// ---- DUTs/Controllers/Band.TcPOU
FUNCTION Band : LREAL
VAR_INPUT
	Value: lreal;
	Target: LREAL;
	Width: LREAL;
END_VAR
VAR
END_VAR

  Band := LimitValue(Value - Target, -Width, Width) / Width;

END_FUNCTION

// ---- DUTs/Controllers/BandLimit.TcPOU
FUNCTION BandLimit : LREAL
VAR_INPUT
	Value: LREAL;
	Target: LREAL;
	Width: LREAL;
	MinValue: LREAL;
	MaxValue: LREAL;
END_VAR
VAR
END_VAR

BandLimit := LimitValue(Band(Value, Target, Width), MinValue, MaxValue);

END_FUNCTION

// ---- DUTs/Controllers/Controller.TcPOU
FUNCTION_BLOCK Controller
VAR_INPUT
	EN: BOOL;
    SP: LREAL;          (* Set point                           *)
    PV: LREAL;          (* Process value                       *)
    p_gain: LREAL;      (* Proportional gain (stiffness)       *)
    i_gain: LREAL;      (* integral gain (windup)              *)
END_VAR
VAR_OUTPUT
	ENO: BOOL;
    CV: LREAL;          (* Control value              *)
END_VAR
VAR
    { Parameters }

    { Calculated values }

    { Local variables}
    integral: LREAL;
    last_error: LREAL;
    last_output: LREAL;
    this_target: LREAL;
    next_target: LREAL;
    ITimer: Timer;    (* Integration timer *)
    LastITime: LINT;
    Timer: Timer;    (* Update timer *)
    MinControl: Timer;
    MaxControl: Timer;
END_VAR

ENO := EN;
IF EN THEN
	Compute();
ELSE
	Reset();	
END_IF

METHOD Compute : BOOL
VAR_INPUT
END_VAR
VAR
  this_error: LREAL;
  this_output: LREAL;
  new_integral: LREAL;
  TimeValue: LINT;

END_VAR
(* the desired PV for this iteration is the value     *)
(* calculated as next_target during the last loop     *)
this_target := next_target;

next_target := SP;

(* the error for the current pass is the difference   *)
(* between the current target and the current PV      *)
this_error := this_target - PV;

{ the new error is added to the integral             }
TimeValue := ITimer.ElapsedTime();
new_integral := integral + i_gain * (this_target - PV) * ((1.0 * LINT_TO_LREAL(TimeValue - LastITime)) / LINT_TO_LREAL(ITimer.TimeoutTime));
LastITime := TimeValue;
IF (new_integral + p_gain * this_error) > 1 THEN
	integral := 1 - p_gain * this_error;
ELSIF (new_integral + p_gain * this_error) < 0 THEN
	integral := -p_gain * this_error;
ELSE
	integral := new_integral;
END_IF;
IF ITimer.Timeout() THEN
	ITimer.Restart();
	LastITime := 0;
END_IF;

(* now that all of the variable terms have been       *)
(* computed they can be multiplied by the appropriate *)
(* coefficients and the resulting products summed     *)
this_output := p_gain * this_error + integral;

last_error := this_error;

(* now check the output value for absolute limits     *)
IF (this_output < 0) THEN
	(* Limit I *)
	if integral < 0 then
		integral := LimitValue(integral, integral - this_output, 0);
	END_IF;
	this_output := 0;
ELSIF (this_output > 1) THEN
	(* Limit I *)
	if integral > 0 then
		integral := LimitValue(integral, 0, integral - (this_output - 1));
	END_IF;
	(* Limit output *)
	this_output := 1;
END_IF;

(* store the new output value to be used as the old   *)
(* output value on the next loop pass                 *)
last_output := this_output;

CV := this_output;
IF Timer.Timeout() THEN
	Timer.Restart();
END_IF;
IF CV > 0.01 THEN
	MinControl.Restart();
END_IF;
IF CV < (1 - 0.01) THEN
	MaxControl.Restart();
END_IF;
END_METHOD

METHOD FB_init : BOOL
VAR_INPUT
	bInitRetains : BOOL; // if TRUE, the retain variables are initialized (warm start / cold start)
	bInCopyCode : BOOL;  // if TRUE, the instance afterwards gets moved into the copy code (online change)
END_VAR
p_gain := 0.5;
i_gain := 0.5;
ITimer.TimeoutTime := 30000;
Timer.TimeoutTime := 1000;
END_METHOD

METHOD Preset : BOOL
VAR_INPUT
	Target: LREAL;
	Control: LREAL;
END_VAR
  last_error := 0;
  last_output := Control;
  next_target := Target;
  this_target := Target;
  ResetIntegral();
  integral := Control;
  CV := Control;
  SP := Target;
END_METHOD

METHOD Reset : BOOL
VAR_INPUT
END_VAR
  ResetIntegral();
  last_error := 0;
  last_output := 0;
  next_target := 0;
  this_target := 0;
  CV := 0;
  SP := 0;
  MinControl.Restart();
  MaxControl.Restart();
END_METHOD

METHOD ResetIntegral : BOOL
VAR_INPUT
END_VAR
  integral := 0;
  ITimer.Restart();
  LastITime := ITimer.ElapsedTime();
END_METHOD

END_FUNCTION_BLOCK

// ---- DUTs/Controllers/InterpolateNewton.TcPOU
FUNCTION_BLOCK InterpolateNewton
VAR_INPUT
	EN: BOOL;
	x: LREAL;
END_VAR
VAR_OUTPUT
	ENO: BOOL;
	y: LREAL;
END_VAR
VAR CONSTANT
	NUM_POINTS: INT := 9;
END_VAR
VAR
	InitDone: BOOL;
	yd: ARRAY [0..NUM_POINTS - 1, 0..NUM_POINTS - 1] OF LREAL;
	i: INT;
END_VAR
VAR PERSISTENT
	xd: ARRAY [0..NUM_POINTS - 1] OF LREAL;
	yv: ARRAY [0..NUM_POINTS - 1] OF LREAL;
END_VAR

IF NOT InitDone THEN
	FOR i := 0 TO NUM_POINTS - 1 DO
		yd[i, 0] := yv[i];
	END_FOR
	DividedDiffTable();
	InitDone := TRUE;
END_IF
y := ApplyFormula(x);
ENO := EN;

METHOD ApplyFormula : LREAL
VAR_INPUT
	Value: LREAL;
END_VAR
VAR
	Sum: LREAL;
	i: INT;
END_VAR
Sum := yd[0, 0];
FOR i := 1 TO NUM_POINTS - 1 DO
	Sum := Sum + ProTerm(i, Value) * yd[0, i];
END_FOR
ApplyFormula := Sum;
END_METHOD

METHOD DividedDiffTable : BOOL
VAR_INPUT
END_VAR
VAR
	i: INT;
	j: int;
END_VAR
FOR i := 1 TO NUM_POINTS - 1 DO
	FOR j := 0 TO NUM_POINTS - i - 1 DO
		IF ABS(xd[j] - xd[i + j]) > 0.00000001 THEN
			yd[j,i] := (yd[j,i - 1] - yd[j + 1,i - 1]) / (xd[j] - xd[i + j]);			
		END_IF
	END_FOR
END_FOR
DividedDiffTable := TRUE;
END_METHOD

METHOD ProTerm : LREAL
VAR_INPUT
	i: INT;
	Value: LREAL;
END_VAR
VAR
	Pro: LREAL;
	j: int;
END_VAR
Pro := 1;
FOR j := 0 TO i - 1 DO
	Pro := Pro * (Value - xd[j]);
END_FOR
ProTerm := Pro;
END_METHOD

END_FUNCTION_BLOCK

// ---- DUTs/Controls/ExtractAirControl.TcPOU
FUNCTION_BLOCK ExtractAirControl
VAR_INPUT
	EN: BOOL;
END_VAR
VAR_OUTPUT
	ENO: BOOL;
END_VAR
VAR
END_VAR

ENO := EN;

END_FUNCTION_BLOCK

// ---- DUTs/Fire/FireDamper.TcPOU
FUNCTION_BLOCK FireDamper EXTENDS Damper
VAR_INPUT
END_VAR
VAR_OUTPUT
END_VAR
VAR
END_VAR

END_FUNCTION_BLOCK

// ---- DUTs/Fire/SmokeDetector.TcPOU
FUNCTION_BLOCK SmokeDetector
VAR_INPUT
	EN: BOOL;
	Input: REFERENCE TO AnalogInput;
	FireAlarm: REFERENCE TO AnalogAlarm;
	ServiceAlarm: REFERENCE TO AnalogAlarm;
END_VAR
VAR_OUTPUT
	ENO: BOOL;
END_VAR
VAR
END_VAR

END_FUNCTION_BLOCK

// ---- DUTs/GreenMaster/IO/GreenMasterAIU.TcPOU
FUNCTION_BLOCK GreenMasterAIU EXTENDS GreenMasterAIU_Base
VAR_INPUT
END_VAR
VAR_OUTPUT
END_VAR
VAR
	IO_AI_09: PressureInput;
	IO_AI_10: PressureInput;
	IO_AI_11: PressureInput;
	IO_AI_12: PressureInput;
	IO_AI_13: PressureInput;
	IO_AI_14: PressureInput;
	IO_AI_15: PressureInput;
	IO_AI_16: PressureInput;
END_VAR


// PAGE AI
IO_AI_09(ProcessError := Globals.IO.AIn.AI17_Error, ProcessValue := Globals.IO.AIn.AI17, Range := 3500); // PressureInput
T_BF1_Error := IO_AI_09.Error;
IO_AI_10(ProcessError := Globals.IO.AIn.AI18_Error, ProcessValue := Globals.IO.AIn.AI18, Range := 3500); // PressureInput
T_BF1 := IO_AI_09.Value;
F_BF1_Error := IO_AI_10.Error;
F_BF1 := IO_AI_10.Value;
IO_AI_11(ProcessError := Globals.IO.AIn.AI19_Error, ProcessValue := Globals.IO.AIn.AI19, Range := 500); // PressureInput
T_BP2_Error := IO_AI_11.Error;
IO_AI_12(ProcessError := Globals.IO.AIn.AI20_Error, ProcessValue := Globals.IO.AIn.AI20, Range := 500); // PressureInput
T_BP2 := IO_AI_11.Value;
F_BP2_Error := IO_AI_12.Error;
F_BP2 := IO_AI_12.Value;
IO_AI_13(ProcessError := Globals.IO.AIn.AI21_Error, ProcessValue := Globals.IO.AIn.AI21, Range := 500); // PressureInput
F_BP3_Error := IO_AI_13.Error;
IO_AI_14(ProcessError := Globals.IO.AIn.AI22_Error, ProcessValue := Globals.IO.AIn.AI22, Range := 500); // PressureInput
F_BP3 := IO_AI_13.Value;
T_BP1_Error := IO_AI_14.Error;
T_BP1 := IO_AI_14.Value;
IO_AI_15(ProcessError := Globals.IO.AIn.AI23_Error, ProcessValue := Globals.IO.AIn.AI23, Range := 500); // PressureInput
F_BP1_Error := IO_AI_15.Error;
IO_AI_16(ProcessError := Globals.IO.AIn.AI24_Error, ProcessValue := Globals.IO.AIn.AI24); // PressureInput
F_BP1 := IO_AI_15.Value;

END_FUNCTION_BLOCK

// ---- DUTs/IO/AnalogSwitch.TcPOU
FUNCTION_BLOCK AnalogSwitch
VAR_INPUT
	EN: BOOL;
	Index: INT;
	Input01: LREAL;
	Input02: LREAL;
	Input03: LREAL;
	Input04: LREAL;
	Input05: LREAL;
	Input06: LREAL;
	Input07: LREAL;
	Input08: LREAL;
END_VAR
VAR_OUTPUT
	ENO: BOOL;
	Output: LREAL;
END_VAR
VAR
END_VAR

END_FUNCTION_BLOCK

// ---- DUTs/ModbusRTU/ModbusWriteWord.TcPOU
FUNCTION_BLOCK ModbusWriteWord EXTENDS ModbusIo
VAR_INPUT
	Value: WORD;
END_VAR
VAR_OUTPUT
END_VAR
VAR
END_VAR

SUPER^();

END_FUNCTION_BLOCK

// ---- DUTs/Parameters/Regulation/DefaultParametersFB.TcPOU
FUNCTION_BLOCK DefaultParametersFB
VAR_INPUT
END_VAR
VAR_OUTPUT
END_VAR
VAR
END_VAR

END_FUNCTION_BLOCK

// ---- DUTs/Parameters/Simulation/SimulateFlow.TcPOU
FUNCTION_BLOCK SimulateFlow
VAR_INPUT
	EN: BOOL;
	SP: LREAL;
	CV: LREAL;
END_VAR
VAR_OUTPUT
	ENO: BOOL;
	Flow: LREAL;
END_VAR
VAR
	Ramp: Ramp;
	FlowFactor: LREAL;
END_VAR

IF EN THEN
	FlowFactor := 1;
	FlowFactor := FlowFactor * MAX(1, CV / 500);
	Ramp(Target := SP * 30000, SpeedUp := 50, SpeedDown := 100, Value => Flow);
END_IF

END_FUNCTION_BLOCK

// ---- DUTs/Parameters/Simulation/SimulationParametersFB.TcPOU
FUNCTION_BLOCK SimulationParametersFB
VAR_INPUT
END_VAR
VAR_OUTPUT
END_VAR
VAR
END_VAR

SimCounter := SimCounter + 1;

END_FUNCTION_BLOCK

// ---- DUTs/Parameters/System/Exercise/ExerciseExternalFireControlParametersFB.TcPOU
FUNCTION_BLOCK ExerciseExternalFireControlParametersFB
VAR_INPUT
END_VAR
VAR_OUTPUT
END_VAR
VAR
END_VAR

END_FUNCTION_BLOCK

// ---- DUTs/Parameters/System/Operation/TimeChannelDayParametersFB.TcPOU
FUNCTION_BLOCK TimeChannelDayParametersFB
VAR_INPUT
END_VAR
VAR_OUTPUT
END_VAR
VAR
END_VAR

END_FUNCTION_BLOCK

// ---- DUTs/System/Supervisor.TcPOU
FUNCTION_BLOCK Supervisor
VAR_INPUT
	EN: BOOL;
	Stop: BOOL;
END_VAR
VAR_OUTPUT
	ENO: BOOL;
END_VAR
VAR
END_VAR
VAR PERSISTENT
END_VAR

ENO := EN AND NOT Stop;

METHOD FB_init : BOOL
VAR_INPUT
	bInitRetains : BOOL; // if TRUE, the retain variables are initialized (warm start / cold start)
	bInCopyCode : BOOL;  // if TRUE, the instance afterwards gets moved into the copy code (online change)
END_VAR
END_METHOD

END_FUNCTION_BLOCK

// ---- DUTs/Utilities/ActuatorMonitor.TcPOU
FUNCTION_BLOCK ActuatorMonitor
VAR_INPUT
	Output: LREAL;
	Input: LREAL;
	Activated: BOOL := TRUE;
	ActivatedError: BOOL := FALSE;
	TimeoutMs: DINT := 30000;
	Treshold: LREAL := 0.1;
END_VAR
VAR_OUTPUT
	Error: BOOL := FALSE;
END_VAR
VAR
	ActivatedSignal: DigitalSignal;
	OutputOnTimer: Timer;
	InputOffTimer: Timer;
END_VAR

// Measure ON time for activation signal
ActivatedSignal(Signal := Activated);

// Measure ON time for output signal
IF Output < Treshold THEN
	OutputOnTimer.Restart();
END_IF

// Measure OFF time for 50% input signal
IF Input >= (Treshold / 2) THEN
	InputOffTimer.Restart();
END_IF

Error := 	(
				(ActivatedSignal.OnTime() > TimeoutMs) AND 
				(OutputOnTimer.ElapsedTime() > TimeoutMs) AND 
				(
					(InputOffTimer.ElapsedTime() > TimeoutMs) OR
					ActivatedError
				)
			);

END_FUNCTION_BLOCK

// ---- DUTs/Utilities/AnalogMultiplexer.TcPOU
FUNCTION_BLOCK AnalogMultiplexer
VAR_INPUT
	bSelect: BOOL;
	iSelect: INT := -1;
	In0: LREAL := 0;
	In1: LREAL := 0;
	In2: LREAL := 0;
	In3: LREAL := 0;
END_VAR
VAR_OUTPUT
	Out: LREAL;
END_VAR
VAR
END_VAR

IF iSelect = -1 THEN
	IF bSelect THEN
		Out := In1;
	ELSE
		Out := In0;
	END_IF
ELSE
	CASE iSelect OF
		0: 	Out := In0;
		1: 	Out := In1;
		2: 	Out := In2;
		3: 	Out := In3;
	END_CASE
END_IF

END_FUNCTION_BLOCK

// ---- DUTs/Utilities/ifc_int.TcPOU
FUNCTION ifc_int : INT
VAR_INPUT
	Condition: BOOL;
	ValueTrue: INT;
	ValueFalse: INT;
END_VAR
VAR
END_VAR

IF Condition THEN
	ifc_int := ValueTrue;
ELSE
	ifc_int := ValueFalse;
END_IF

END_FUNCTION

// ---- DUTs/Utilities/BOOL_BMUX.TcPOU
FUNCTION BOOL_BMUX : BOOL
VAR_INPUT
	B: BOOL;
	X: BOOL;
	Y: BOOL
;
END_VAR
VAR
END_VAR

IF NOT B THEN
	BOOL_BMUX := X;
ELSE
	BOOL_BMUX := Y;
END_IF

END_FUNCTION

// ---- DUTs/Utilities/EMA.TcPOU
FUNCTION_BLOCK EMA
VAR_INPUT
	NewValue: LREAL;
END_VAR
VAR_OUTPUT
	Value: LREAL;
END_VAR
VAR
	Weight: LREAL;
END_VAR

Value := Weight * NewValue + (1 - Weight) * Value;

METHOD FB_init : BOOL
VAR_INPUT
	bInitRetains : BOOL; // if TRUE, the retain variables are initialized (warm start / cold start)
	bInCopyCode : BOOL;  // if TRUE, the instance afterwards gets moved into the copy code (online change)
END_VAR
SetSampleCount(100);
END_METHOD

METHOD SetSampleCount : BOOL
VAR_INPUT
	n: int;
END_VAR
Weight := 2.0 / (1.0 + n);
END_METHOD

METHOD SetValue : BOOL
VAR_INPUT
	NewValue: LREAL;
END_VAR
Value := NewValue;
END_METHOD

END_FUNCTION_BLOCK

// ---- DUTs/Utilities/GetBit.TcPOU
FUNCTION GetBit : BOOL
VAR_INPUT
	Value: ULINT;
	BitNr: INT;
END_VAR
VAR
END_VAR

GetBit := (Value AND SHL(INT_TO_ULINT(1), BitNr)) <> 0;

END_FUNCTION

// ---- DUTs/Utilities/PulseCounter.TcPOU
FUNCTION_BLOCK PulseCounter
VAR_INPUT
	FM: BOOL;
END_VAR
VAR_OUTPUT
	Flow: LREAL;
	PulseCounter: LINT;
END_VAR
VAR
	Tmp: BOOL;
	Now: LINT;
	Last_FM: BOOL;
	LastTime: LINT;
	FilteredFlow: EMA;
	Pulse: BOOL;
	LastPulseLength: LINT;
END_VAR

Tmp := FM;
Now := GetTickCount();
Pulse := (Tmp AND (Tmp <> Last_FM)); 
IF Pulse THEN
	PulseCounter := PulseCounter + 1;
	LastPulseLength := Now - LastTime;
	IF (Now - LastTime) > 0 THEN
		FilteredFlow(NewValue := 3.6 / (LINT_TO_LREAL(Now - LastTime) / 1000.0));
	END_IF
	LastTime := Now;
END_IF
Last_FM := Tmp;
IF (Now - LastTime) > (2 * LastPulseLength) THEN
	IF (Now - LastTime) > 0 THEN
		FilteredFlow(NewValue := 3.6 / (LINT_TO_LREAL(Now - LastTime) / 1000.0));
	END_IF
END_IF
IF (Now - LastTime) > 30000 THEN
	FilteredFlow.SetValue(0);
END_IF
Flow := FilteredFlow.Value;

METHOD FB_init : BOOL
VAR_INPUT
	bInitRetains : BOOL; // if TRUE, the retain variables are initialized (warm start / cold start)
	bInCopyCode : BOOL;  // if TRUE, the instance afterwards gets moved into the copy code (online change)
END_VAR
FilteredFlow.SetSampleCount(5);
END_METHOD

END_FUNCTION_BLOCK

// ---- DUTs/Utilities/PWM.TcPOU
FUNCTION_BLOCK PWM
VAR_INPUT
END_VAR
VAR_OUTPUT
END_VAR
VAR
	Timer: Timer;
	CurrentDutyCycle: LREAL;
	FPeriod: LREAL;
	FDutyCycle: LREAL;
	FMinValue: LREAL := 0.05; // 5% / 95% min/max value	
END_VAR

PROPERTY DutyCycle : LREAL
GET
DutyCycle := CurrentDutyCycle;
END_GET
SET
VAR
	TimeValue: lreal;	
END_VAR
TimeValue := DutyCycle * Period;
IF (TimeValue < MinValue) THEN
	FDutyCycle := 0;
ELSIF (TimeValue > (Period - MinValue)) THEN
	FDutyCycle := 1;
else
	FDutyCycle := DutyCycle;
END_IF
END_SET
END_PROPERTY

PROPERTY MinValue : LREAL
GET
MinValue := FMinValue;
END_GET
SET
FMinValue := MinValue;
END_SET
END_PROPERTY

PROPERTY Period : LREAL
GET
Period := FPeriod;
END_GET
SET
IF FPeriod <> Period THEN
	FPeriod := Period;
	CurrentDutyCycle := DutyCycle;
	Timer.Restart();
END_IF;
END_SET
END_PROPERTY

METHOD State : BOOL
VAR_INPUT
END_VAR
VAR
	ElapsedTime: LINT;
	Res: BOOL;
END_VAR
ElapsedTime := Timer.ElapsedTime();
IF (ElapsedTime > LREAL_TO_LINT(Period * 1000)) THEN
	ElapsedTime := TRUNC(Period * 1000);
END_IF
Res := ElapsedTime <= LREAL_TO_LINT(CurrentDutyCycle * Period * 1000);
IF (ElapsedTime >= LREAL_TO_LINT(Period * 1000)) THEN
	Timer.Restart();
	CurrentDutyCycle := FDutyCycle;
END_IF;
State := Res;
END_METHOD

END_FUNCTION_BLOCK

// ---- DUTs/Utilities/LREAL_TO_WORD_SAFE.TcPOU
FUNCTION LREAL_TO_WORD_SAFE : WORD
VAR_INPUT
	Value: LREAL;
END_VAR
VAR
END_VAR

LREAL_TO_WORD_SAFE := TO_WORD(TO_LINT(Value));

END_FUNCTION

// ---- DUTs/Utilities/SetBit.TcPOU
FUNCTION SetBit : ULINT
VAR_INPUT
	Value: ULINT;
	BitNr: INT;
	State: BOOL;
END_VAR
VAR
END_VAR

IF State THEN
	SetBit := (Value AND (NOT SHL(INT_TO_ULINT(1), BitNr))) OR SHL(INT_TO_ULINT(1), BitNr);
ELSE
	SetBit := (Value AND (NOT SHL(INT_TO_ULINT(1), BitNr)));
END_IF

END_FUNCTION

// ---- DUTs/Valves/BaseValve.TcPOU
FUNCTION_BLOCK BaseValve
VAR_INPUT
	Open: REFERENCE TO BOOL;
	IsOpen: REFERENCE TO BOOL;
	IsClosed: REFERENCE TO BOOL;
END_VAR
VAR_OUTPUT
END_VAR
VAR
END_VAR

END_FUNCTION_BLOCK

// ---- DUTs/Valves/Valve.TcPOU
FUNCTION_BLOCK Valve EXTENDS BaseValve
VAR_INPUT
	IO_Open: REFERENCE TO DigitalOutput;
	IO_FB1, IO_FB2: REFERENCE TO DigitalInput;
END_VAR
VAR_OUTPUT
END_VAR
VAR
	ValveMonitor: ValveMonitor; 
	Error: BOOL;
END_VAR

ValveMonitor(Valve := Open, FB1 := IsOpen, FB2 := IsClosed);
Error := ValveMonitor.Error;

END_FUNCTION_BLOCK

// ---- DUTs/Valves/ValveMonitor.TcPOU
FUNCTION_BLOCK ValveMonitor
VAR_INPUT
	Valve: BOOL;	// Valve DO
	FB1: BOOL;		// Open DI
	FB2: BOOL;		// Closed DI
	Timeout: TIME;
END_VAR
VAR_OUTPUT
	Error: BOOL;
END_VAR
VAR
	ValveSignal: DigitalSignal;
	ValveOpenTimer: Timer;
	ValveClosedTimer: Timer;
END_VAR

ValveSignal(Signal := Valve);
IF Main.GreenMaster.GetParameters().System.Operation.State <> SystemStates.Run THEN
	Error := FALSE;
ELSE
	Error := ((ValveSignal.OnTime() > TO_LINT(T#30S)) AND (NOT FB1)) OR
		((ValveSignal.OffTime() > TO_LINT(T#30S)) AND (NOT FB2));	
END_IF

END_FUNCTION_BLOCK

// ---- DUTs/Ventilation/FB_GM_NIGHTCOOL.TcPOU
FUNCTION_BLOCK FB_GM_NIGHTCOOL
VAR_INPUT
	bDayOperation						: BOOL; // Normal daytime operation
	rNormalSAPressure					: REAL; // Normal daytime operation setpoint for supply air pressure
	rNormalEAPressure					: REAL; // Normal daytime operation setpoint for extract air pressure
	rNormalTemperature					: REAL; // Normal daytime operation setpoint for supply air temperature
END_VAR
VAR_OUTPUT
	bStartNightcool						: BOOL; // Starts GreenMaster in nightcool	
	rSAPressure							: REAL; // Supply air pressure when nightcooling is active
	rEAPressure							: REAL;	// Extract air pressure when nightcooling is active
	rSATemperature						: REAL; // Supply air temperature when nightcooling is active
	bNightCoolActive					: BOOL; // Nightcooling is active
	rExtractAirTemperature				: REAL;	// Saftey input
END_VAR
VAR PERSISTENT
	rSupplyPressure						: REAL; // Supply air pressure when nightcooling is active
	rExtractPressure					: REAL; // Extract air pressure when nightcooling is active
	rSupplyTemperature					: REAL; // Supply air temperature when nightcooling is active
	bCMD								: BOOL; // Start nightcooling from HMI
END_VAR

// Om vi kör nattkyla så har vi nya börvärden
IF bStartNightcool THEN
	rSAPressure := rSupplyPressure;   // New SA Pressure setpoint
	rEAPressure := rExtractPressure;  // New EA Pressire setpint
	rSATemperature :=  MAX (13,rSupplyTemperature); // New SA temperature setpoint with limit 
	bNightCoolActive :=TRUE;
ELSE
	rSAPressure := rNormalSAPressure;
    rEAPressure := rNormalEAPressure;
    rSATemperature := rNormalTemperature;
	bNightCoolActive :=FALSE;
END_IF

// Sätter utgång för att starta aggregat (med säkerhetsfunktion då frånluftstemperatur blir för låg)
IF NOT bDayOperation AND NOT(rExtractAirTemperature < 17) THEN
	IF bCMD THEN
		bStartNightcool := TRUE;
	ELSE
		bStartNightcool := FALSE;
	END_IF
ELSE 
	bStartNightcool := FALSE;
END_IF

END_FUNCTION_BLOCK

// ---- POUs/AdsWriteVariable.TcPOU
FUNCTION_BLOCK AdsWriteVariable
VAR_INPUT
	NetID: STRING := '';
	Name: STRING;
	EN: BOOL;
	Source: PVOID;
END_VAR
VAR_OUTPUT
	ENO: BOOL;
END_VAR
VAR
	PLC_ReadSymInfoByName: PLC_ReadSymInfoByName;
	ADSWRITE: ADSWRITE;
	State : INT := 0;
END_VAR

CASE State OF
0:
	IF EN THEN
		State := 1;
	END_IF
1:	
	PLC_ReadSymInfoByName(
		NETID := NetID, 
		PORT := 851, 
		SYMNAME := Name,
		TMOUT := T#5S,
		START := TRUE
	);
	State := 2;
2:
	PLC_ReadSymInfoByName();
	IF NOT PLC_ReadSymInfoByName.BUSY THEN
		PLC_ReadSymInfoByName(START := FALSE);
		ADSWRITE(
			NETID:= '',
			PORT:= 851,
			IDXGRP:= PLC_ReadSymInfoByName.SYMINFO.idxGroup,
			IDXOFFS:= PLC_ReadSymInfoByName.SYMINFO.idxOffset,
			LEN:= SIZEOF(PLC_ReadSymInfoByName.SYMINFO.byteSize),
			SRCADDR:= Source,
			WRITE:= TRUE,
			TMOUT:= T#5S,
		);
		State := 3;		
	END_IF
	IF NOT EN THEN
		ADSWRITE(WRITE := FALSE);
		ENO := FALSE;
		State := 0;
	END_IF
3:
	ADSWRITE();
	IF NOT ADSWRITE.BUSY THEN
		ENO := TRUE;
		ADSWRITE(WRITE := FALSE);
	END_IF
	IF NOT EN THEN
		ADSWRITE(WRITE := FALSE);
		ENO := FALSE;
		State := 0;
	END_IF
END_CASE

END_FUNCTION_BLOCK

// ---- POUs/SimpleTimeChannel.TcPOU
FUNCTION_BLOCK SimpleTimeChannel
VAR_INPUT
	EN: BOOL;
END_VAR
VAR_OUTPUT
	ENO: BOOL;
END_VAR
VAR
	LocalSystemTime: FB_LocalSystemTime;
	Active: BOOL;
	InitDone: bool;
END_VAR

IF NOT InitDone THEN
	EN := TRUE;
	InitDone := TRUE;
END_IF
LocalSystemTime(bEnable := TRUE);
IF LocalSystemTime.bValid THEN
	Active := (NOT EN) OR ((LocalSystemTime.systemTime.wHour > 5 AND LocalSystemTime.systemTime.wHour < 20) OR
		(LocalSystemTime.systemTime.wHour = 5 AND LocalSystemTime.systemTime.wMinute >= 30)); 
END_IF

ENO := EN AND Active;

END_FUNCTION_BLOCK

// ---- POUs/AdsReadVariable.TcPOU
FUNCTION_BLOCK AdsReadVariable
VAR_INPUT
	NetID: STRING := '';
	Name: STRING;
	EN: BOOL;
	Destination: PVOID;
END_VAR
VAR_OUTPUT
	ENO: BOOL;
END_VAR
VAR
	PLC_ReadSymInfoByName: PLC_ReadSymInfoByName;
	ADSREADEX: ADSREADEX;
	State : INT := 0;
END_VAR

CASE State OF
0:
	IF EN THEN
		State := 1;
	END_IF
1:	
	PLC_ReadSymInfoByName(
		NETID := NetID, 
		PORT := 851, 
		SYMNAME := Name,
		TMOUT := T#5S,
		START := TRUE
	);
	State := 2;
2:
	PLC_ReadSymInfoByName();
	IF NOT PLC_ReadSymInfoByName.BUSY THEN
		PLC_ReadSymInfoByName(START := FALSE);
		ADSREADEX(
			NETID:= '',
			PORT:= 851,
			IDXGRP:= PLC_ReadSymInfoByName.SYMINFO.idxGroup,
			IDXOFFS:= PLC_ReadSymInfoByName.SYMINFO.idxOffset,
			LEN:= SIZEOF(PLC_ReadSymInfoByName.SYMINFO.byteSize),
			DESTADDR:= Destination,
			READ:= TRUE,
			TMOUT:= T#5S,
		);
		State := 3;		
	END_IF
	IF NOT EN THEN
		ADSREADEX(READ := FALSE);
		ENO := FALSE;
		State := 0;
	END_IF
3:
	ADSREADEX();
	IF NOT ADSREADEX.BUSY THEN
		ENO := TRUE;
		ADSREADEX(READ := FALSE);
	END_IF
	IF NOT EN THEN
		ADSREADEX(READ := FALSE);
		ENO := FALSE;
		State := 0;
	END_IF
END_CASE

END_FUNCTION_BLOCK
